// TIA Portal V17 export
// export: Created 2025-03-12T15:36:02.631237Z, ExportSetting WithDefaults, DisplayName Totally Integrated Automation Portal, DisplayVersion V17 Update 8, DisplayName TIA Portal Openness, DisplayVersion V17 Update 8, DisplayName TIA Portal Version Control Interface, DisplayVersion V17, DisplayName SINAMICS Startdrive Advanced, DisplayVersion V17 SP2, DisplayName SINAMICS Startdrive G110M, G120, G120C, G120D, G120P, G115D, DisplayVersion V17 SP2, DisplayName SINAMICS Startdrive G130, G150, S120, S150, SINAMICS MV, S210, DisplayVersion V17 SP2, DisplayName STEP 7 Professional, DisplayVersion V17 Update 8, DisplayName SINUMERIK ONE STEP 7 Toolbox, DisplayVersion V17 Update 12, DisplayName SINUMERIK 840D sl STEP 7 Toolbox, DisplayVersion V17 Update 12, DisplayName STEP 7 Safety, DisplayVersion V17 Update 6, DisplayName WinCC Advanced, DisplayVersion V17 Update 8
DATA_BLOCK "DB2392_POWER_METER"   // DB2392
{ S7_Optimized_Access := 'FALSE'; DB_Accessible_From_OPC_UA := 'FALSE' }
AUTHOR : ETXETAR
VERSION : 1.0
// stored: AutoNumber false, DBAccessibleFromOPCUA false, DBAccessibleFromWebserver true, IsOnlyStoredInLoadMemory false, IsWriteProtectedInAS false
   VAR RETAIN
      VOLTAGE_L1_N : Real;   // VOLTAGE L1 N
      VOLTAGE_L2_N : Real;   // VOLTAGE L2 N
      VOLTAGE_L3_N : Real;   // VOLTAGE L3 N
      VOLTAGE_L1_L2 : Real;   // VOLTAGE L1-L2
      VOLTAGE_L2_L3 : Real;   // VOLTAGE L2-L3
      VOLTAGE_L3_L1 : Real;   // VOLTAGE L3-L1
      CURRENT_L1 : Real;   // CURRENT L1
      CURRENT_L2 : Real;   // CURRENT L2
      CURRENT_L3 : Real;   // CURRENT L3
      ACTIVE_POWER_L1 : Real;   // ACTIVE POWER L1
      ACTIVE_POWER_L2 : Real;   // ACTIVE POWER L2
      ACTIVE_POWER_L3 : Real;   // ACTIVE POWER L3
      ACTIVE_ENERGY_IMPORT : Real;   // ACTIVE ENERGY IMPORT
      TOTAL_ACTIVE_POWER : Real;   // TOTAL ACTIVE POWER
      TOTAL_APPARENT_FACTOR : Real;   // TOTAL APPARENT FACTOR
      TOTAL_REACTIVE_POWER : Real;   // TOTAL REACTIVE POWER
      TOTAL_POWER_FACTOR : Real;   // TOTAL POWER FACTOR
      LINE_FREQUENCY : Real;   // LINE FRECUENCY
      CURRENT_UPPER_LIMIT_A : Real;   // CURRENT UPPER LIMIT A
      VOLTAGE_UPPER_LIMIT_V : Real;   // VOLTAGE UPPER LIMIT V
      VOLTAGE_LOWER_LIMIT_V : Real;   // VOLTAGE LOWER LIMIT V
      IMPORT_DAY : Real;   // IMPORT DAY
      IMPORT_DAY_AUX : Real;   // IMPORT DAY AUXILIARY
      IMPORT_DAY_1 : Real;   // IMPORT DAY 1
      IMPORT_DAY_2 : Real;   // IMPORT DAY 2
      IMPORT_DAY_3 : Real;   // IMPORT DAY 3
      IMPORT_DAY_4 : Real;   // IMPORT DAY 4
      IMPORT_DAY_5 : Real;   // IMPORT DAY 5
      IMPORT_DAY_6 : Real;   // IMPORT DAY 6
      IMPORT_DAY_7 : Real;   // IMPORT DAY 7
      IMPORT_DAY_8 : Real;   // IMPORT DAY 8
      IMPORT_DAY_9 : Real;   // IMPORT DAY 9
      IMPORT_DAY_10 : Real;   // IMPORT DAY 10
      HMI_CURRENT_UPPER_LIMIT_LED : Bool;   // HMI CURRENT UPPER LIMIT LED
      HMI_VOLTAGE_UPPER_LIMIT_LED : Bool;   // HMI VOLTAGE UPPER LIMIT LED
      HMI_VOLTAGE_LOWER_LIMIT_LED : Bool;   // HMI VOLTAGE LOWER LIMIT LED
      CURRENT_UPPER_LIMIT_FAULT : Bool;   // CURRENT UPPER LIMIT ALARM
      VOLTAGE_UPPER_LIMIT_FAULT : Bool;   // VOLTAGE UPPER LIMIT ALARM
      VOLTAGE_LOWER_LIMIT_FAULT : Bool;   // VOLTAGE LOWER LIMIT ALARM
      "DATE" : Byte;   // DATE
      SYSTEM_YEAR : Byte;   // SYSTEM YEAR
      SYSTEM_MONTH : Byte;   // SYSTEM MONTH
      SYSTEM_DATE : Byte;   // SYSTEM DATE
      SYSTEM_HOUR : Byte;   // SYSTEM HOUR
      SYSTEM_MINUTE : Byte;   // SYSTEM MINUTE
      SYSTEM_SECOND : Byte;   // SYSTEM SECOND
   END_VAR
BEGIN
END_DATA_BLOCK
